# EPICS substitutions: motorExApp/Db/NoMPF_MX.substitutions
file basic_motor.db
{
pattern
{P,     N,  M,      DTYP,         C,  S,  DESC,          EGU,      DIR,  VELO,  VBAS,  ACCL,  BDST,  BVEL,  BACC,  MRES,  PREC,  DHLM,  DLLM,  INIT}
{rls:,  1,  m$(N),  "MXmotor",    0,  0,  "motor $(N)",  degrees,  Pos,  1,     .1,    .2,    0,     1,     .2,    0.01,  5,     100,   -100,  ""}
}
